PROGRAM MAIN
VAR
END_VAR

"I trigger a build error";

END_PROGRAM

(* stored: Version 1.1.0.1, ProductVersion 3.1.4024.11
   POU MAIN: Id {7501c181-3edf-4c69-84ec-22f09e2dbfb3}, SpecialFunc None *)
